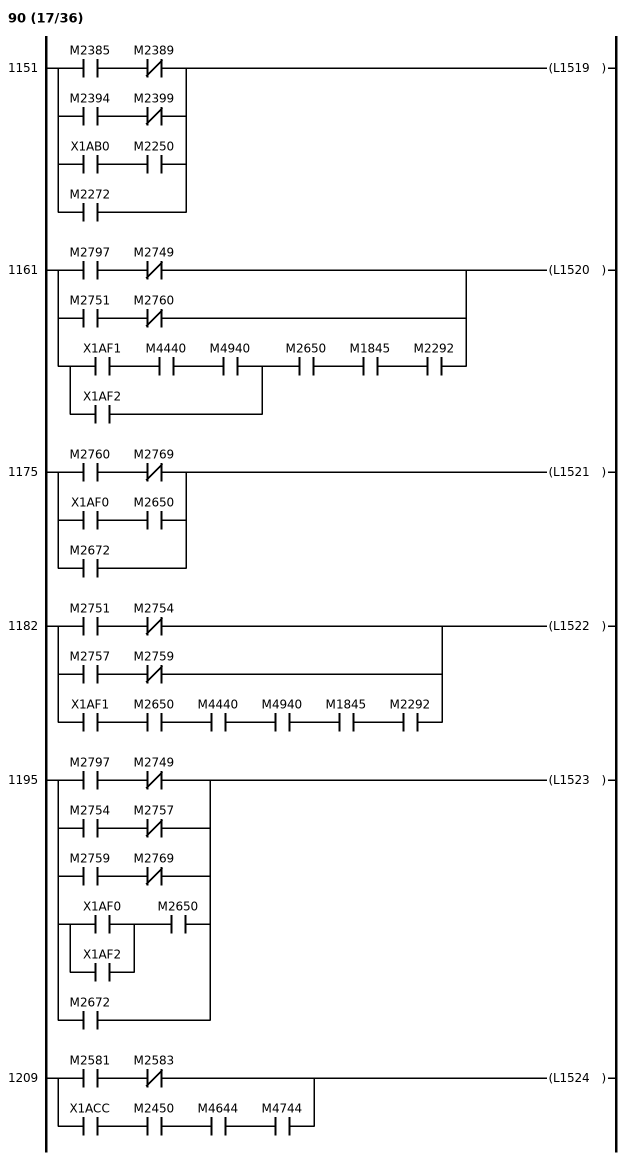
1151  LD      M2385
      ANI     M2389
      LD      M2394
      ANI     M2399
      ORB
      LD      X1AB0
      AND     M2250
      ORB
      OR      M2272
      OUT     L1519
1161  LD      M2797
      ANI     M2749
      LD      M2751
      ANI     M2760
      ORB
      LD      X1AF1
      AND     M4440
      AND     M4940
      OR      X1AF2
      AND     M2650
      AND     M1845
      AND     M2292
      ORB
      OUT     L1520
1175  LD      M2760
      ANI     M2769
      LD      X1AF0
      AND     M2650
      ORB
      OR      M2672
      OUT     L1521
1182  LD      M2751
      ANI     M2754
      LD      M2757
      ANI     M2759
      ORB
      LD      X1AF1
      AND     M2650
      AND     M4440
      AND     M4940
      AND     M1845
      AND     M2292
      ORB
      OUT     L1522
1195  LD      M2797
      ANI     M2749
      LD      M2754
      ANI     M2757
      ORB
      LD      M2759
      ANI     M2769
      ORB
      LD      X1AF0
      OR      X1AF2
      AND     M2650
      ORB
      OR      M2672
      OUT     L1523
1209  LD      M2581
      ANI     M2583
      LD      X1ACC
      AND     M2450
      AND     M4644
      AND     M4744
      ORB
      OUT     L1524
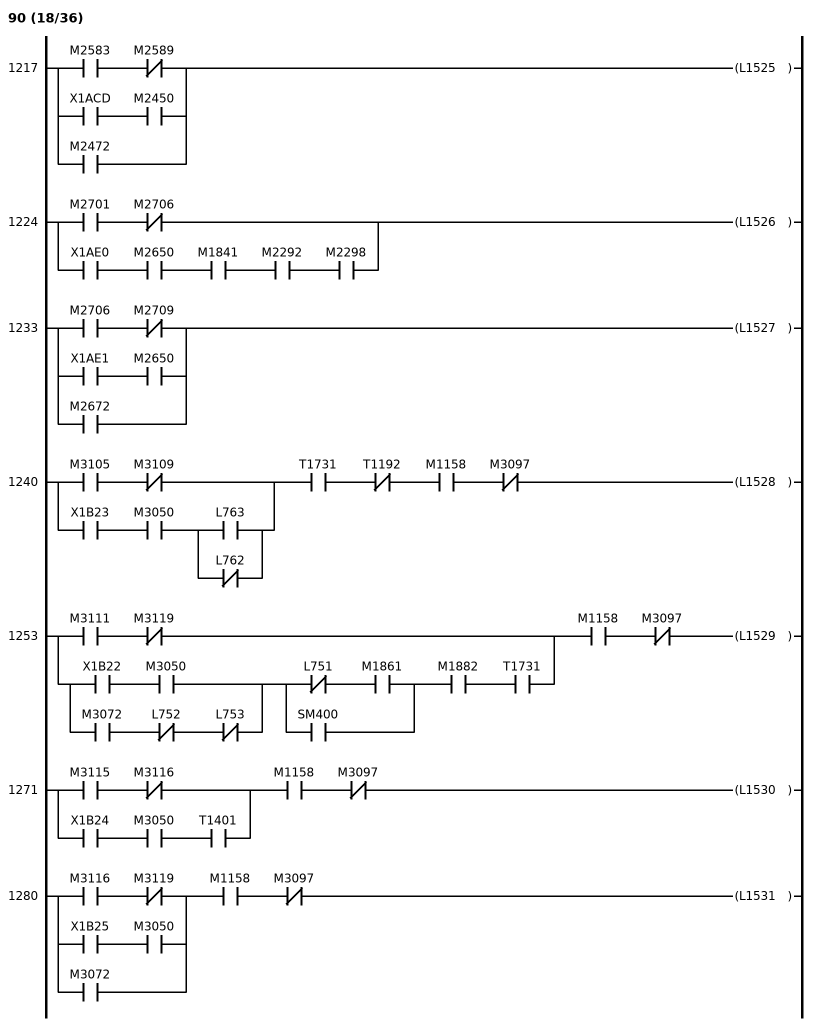
1217  LD      M2583
      ANI     M2589
      LD      X1ACD
      AND     M2450
      ORB
      OR      M2472
      OUT     L1525
1224  LD      M2701
      ANI     M2706
      LD      X1AE0
      AND     M2650
      AND     M1841
      AND     M2292
      AND     M2298
      ORB
      OUT     L1526
1233  LD      M2706
      ANI     M2709
      LD      X1AE1
      AND     M2650
      ORB
      OR      M2672
      OUT     L1527
1240  LD      M3105
      ANI     M3109
      LD      X1B23
      AND     M3050
      LD      L763
      ORI     L762
      ANB
      ORB
      AND     T1731
      ANI     T1192
      AND     M1158
      ANI     M3097
      OUT     L1528
1253  LD      M3111
      ANI     M3119
      LD      X1B22
      AND     M3050
      LD      M3072
      ANI     L752
      ANI     L753
      ORB
      LDI     L751
      AND     M1861
      OR      SM400
      ANB
      AND     M1882
      AND     T1731
      ORB
      AND     M1158
      ANI     M3097
      OUT     L1529
1271  LD      M3115
      ANI     M3116
      LD      X1B24
      AND     M3050
      AND     T1401
      ORB
      AND     M1158
      ANI     M3097
      OUT     L1530
1280  LD      M3116
      ANI     M3119
      LD      X1B25
      AND     M3050
      ORB
      OR      M3072
      AND     M1158
      ANI     M3097
      OUT     L1531
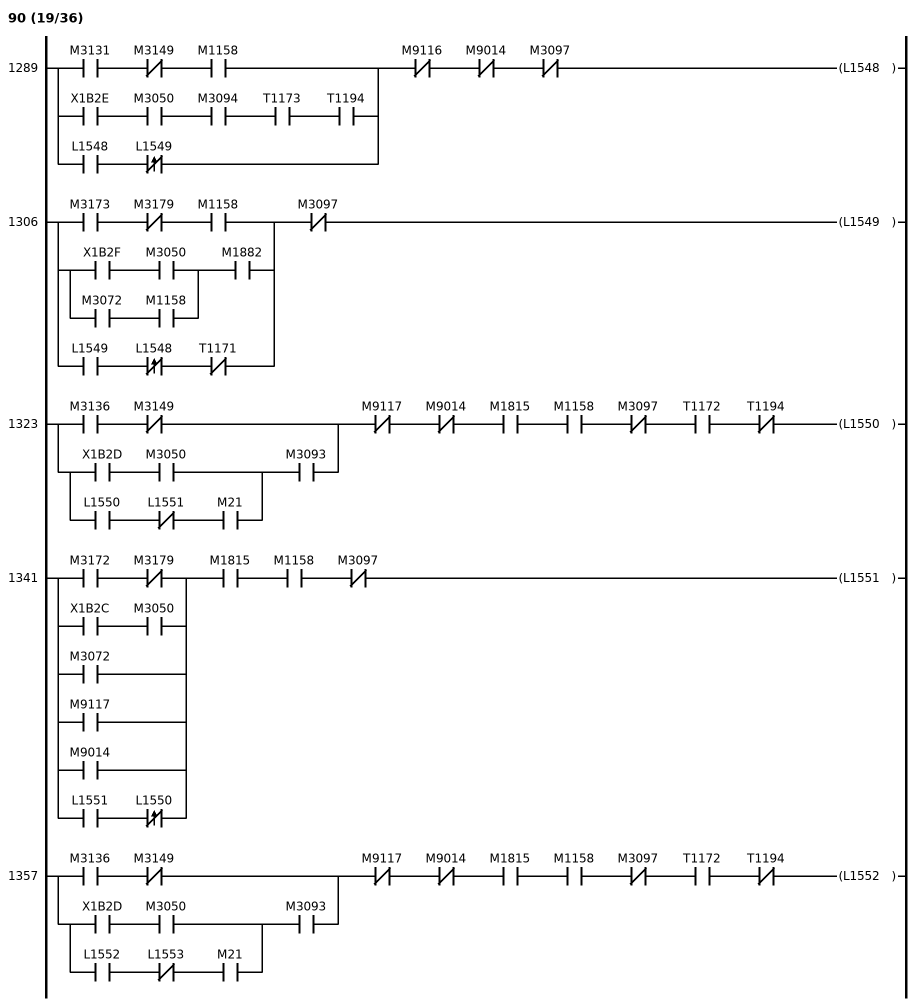
1289  LD      M3131
      ANI     M3149
      AND     M1158
      LD      X1B2E
      AND     M3050
      AND     M3094
      AND     T1173
      AND     T1194
      ORB
      LD      L1548
      ANDPI   L1549
      ORB
      ANI     M9116
      ANI     M9014
      ANI     M3097
      OUT     L1548
1306  LD      M3173
      ANI     M3179
      AND     M1158
      LD      X1B2F
      AND     M3050
      LD      M3072
      AND     M1158
      ORB
      AND     M1882
      ORB
      LD      L1549
      ANDPI   L1548
      ANI     T1171
      ORB
      ANI     M3097
      OUT     L1549
1323  LD      M3136
      ANI     M3149
      LD      X1B2D
      AND     M3050
      LD      L1550
      ANI     L1551
      AND     M21
      ORB
      AND     M3093
      ORB
      ANI     M9117
      ANI     M9014
      AND     M1815
      AND     M1158
      ANI     M3097
      AND     T1172
      ANI     T1194
      OUT     L1550
1341  LD      M3172
      ANI     M3179
      LD      X1B2C
      AND     M3050
      ORB
      OR      M3072
      OR      M9117
      OR      M9014
      LD      L1551
      ANDPI   L1550
      ORB
      AND     M1815
      AND     M1158
      ANI     M3097
      OUT     L1551
1357  LD      M3136
      ANI     M3149
      LD      X1B2D
      AND     M3050
      LD      L1552
      ANI     L1553
      AND     M21
      ORB
      AND     M3093
      ORB
      ANI     M9117
      ANI     M9014
      AND     M1815
      AND     M1158
      ANI     M3097
      AND     T1172
      ANI     T1194
      OUT     L1552
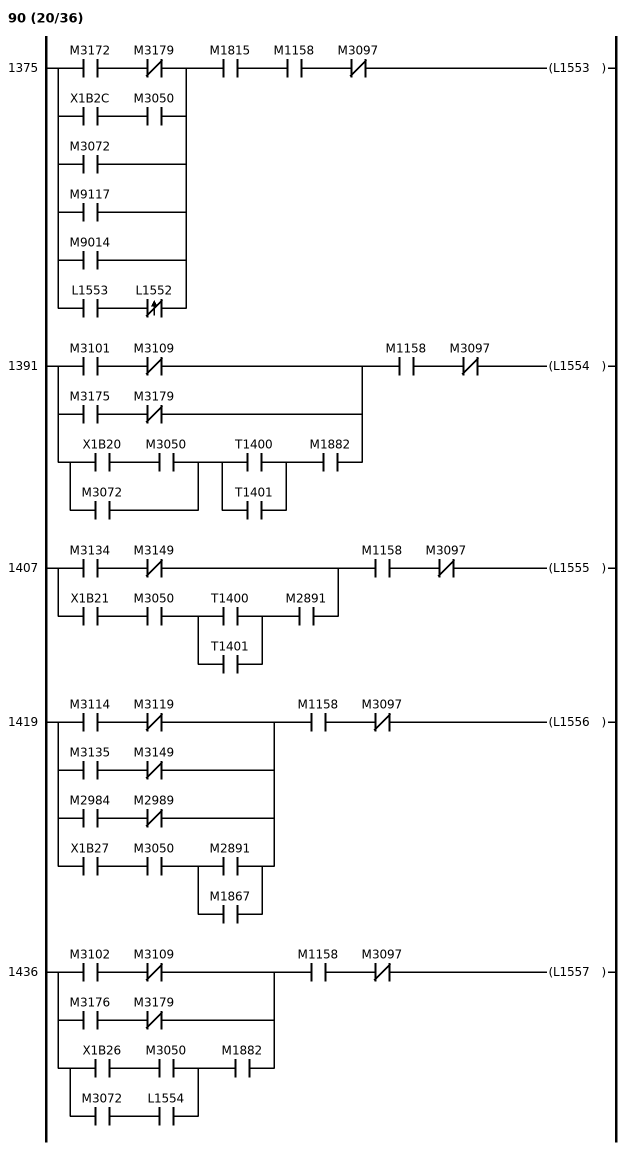
1375  LD      M3172
      ANI     M3179
      LD      X1B2C
      AND     M3050
      ORB
      OR      M3072
      OR      M9117
      OR      M9014
      LD      L1553
      ANDPI   L1552
      ORB
      AND     M1815
      AND     M1158
      ANI     M3097
      OUT     L1553
1391  LD      M3101
      ANI     M3109
      LD      M3175
      ANI     M3179
      ORB
      LD      X1B20
      AND     M3050
      OR      M3072
      LD      T1400
      OR      T1401
      ANB
      AND     M1882
      ORB
      AND     M1158
      ANI     M3097
      OUT     L1554
1407  LD      M3134
      ANI     M3149
      LD      X1B21
      AND     M3050
      LD      T1400
      OR      T1401
      ANB
      AND     M2891
      ORB
      AND     M1158
      ANI     M3097
      OUT     L1555
1419  LD      M3114
      ANI     M3119
      LD      M3135
      ANI     M3149
      ORB
      LD      M2984
      ANI     M2989
      ORB
      LD      X1B27
      AND     M3050
      LD      M2891
      OR      M1867
      ANB
      ORB
      AND     M1158
      ANI     M3097
      OUT     L1556
1436  LD      M3102
      ANI     M3109
      LD      M3176
      ANI     M3179
      ORB
      LD      X1B26
      AND     M3050
      LD      M3072
      AND     L1554
      ORB
      AND     M1882
      ORB
      AND     M1158
      ANI     M3097
      OUT     L1557
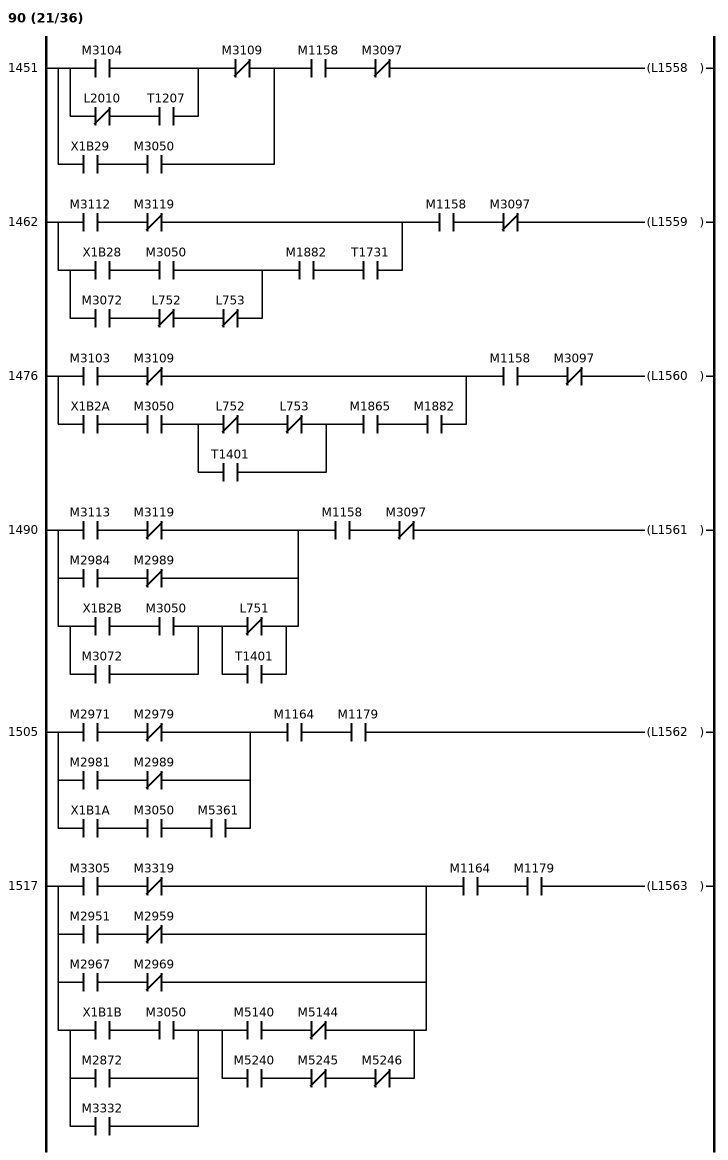
1451  LD      M3104
      LDI     L2010
      AND     T1207
      ORB
      ANI     M3109
      LD      X1B29
      AND     M3050
      ORB
      AND     M1158
      ANI     M3097
      OUT     L1558
1462  LD      M3112
      ANI     M3119
      LD      X1B28
      AND     M3050
      LD      M3072
      ANI     L752
      ANI     L753
      ORB
      AND     M1882
      AND     T1731
      ORB
      AND     M1158
      ANI     M3097
      OUT     L1559
1476  LD      M3103
      ANI     M3109
      LD      X1B2A
      AND     M3050
      LDI     L752
      ANI     L753
      OR      T1401
      ANB
      AND     M1865
      AND     M1882
      ORB
      AND     M1158
      ANI     M3097
      OUT     L1560
1490  LD      M3113
      ANI     M3119
      LD      M2984
      ANI     M2989
      ORB
      LD      X1B2B
      AND     M3050
      OR      M3072
      LDI     L751
      OR      T1401
      ANB
      ORB
      AND     M1158
      ANI     M3097
      OUT     L1561
1505  LD      M2971
      ANI     M2979
      LD      M2981
      ANI     M2989
      ORB
      LD      X1B1A
      AND     M3050
      AND     M5361
      ORB
      AND     M1164
      AND     M1179
      OUT     L1562
1517  LD      M3305
      ANI     M3319
      LD      M2951
      ANI     M2959
      ORB
      LD      M2967
      ANI     M2969
      ORB
      LD      X1B1B
      AND     M3050
      OR      M2872
      OR      M3332
      LD      M5140
      ANI     M5144
      LD      M5240
      ANI     M5245
      ANI     M5246
      ORB
      ANB
      ORB
      AND     M1164
      AND     M1179
      OUT     L1563
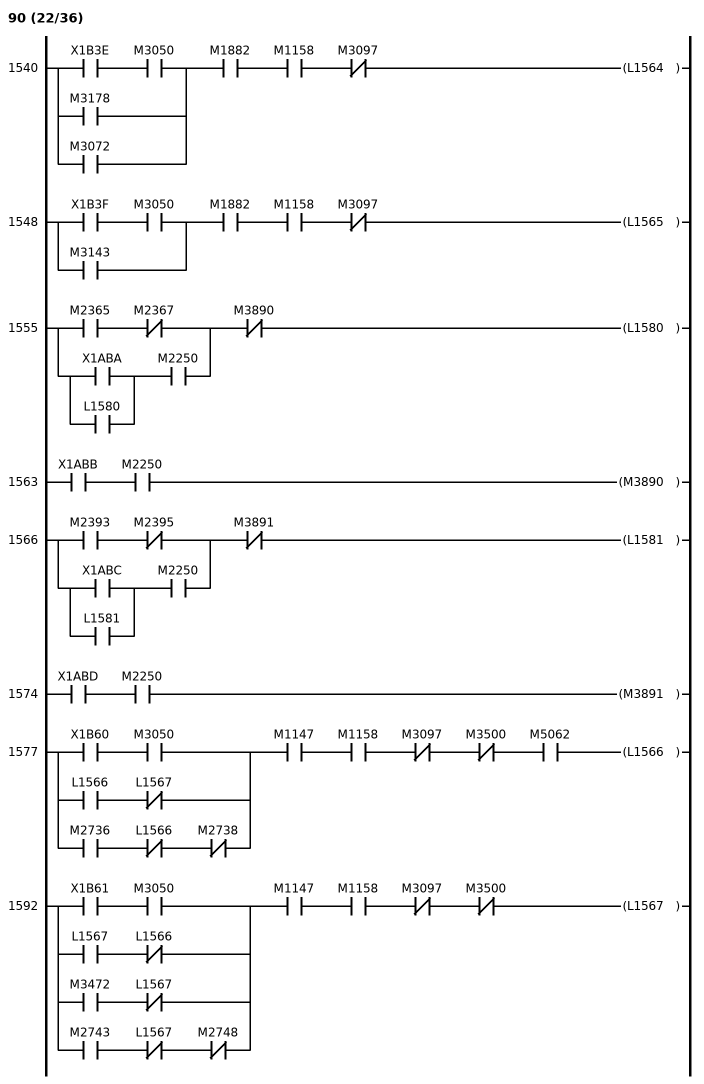
1540  LD      X1B3E
      AND     M3050
      OR      M3178
      OR      M3072
      AND     M1882
      AND     M1158
      ANI     M3097
      OUT     L1564
1548  LD      X1B3F
      AND     M3050
      OR      M3143
      AND     M1882
      AND     M1158
      ANI     M3097
      OUT     L1565
1555  LD      M2365
      ANI     M2367
      LD      X1ABA
      OR      L1580
      AND     M2250
      ORB
      ANI     M3890
      OUT     L1580
1563  LD      X1ABB
      AND     M2250
      OUT     M3890
1566  LD      M2393
      ANI     M2395
      LD      X1ABC
      OR      L1581
      AND     M2250
      ORB
      ANI     M3891
      OUT     L1581
1574  LD      X1ABD
      AND     M2250
      OUT     M3891
1577  LD      X1B60
      AND     M3050
      LD      L1566
      ANI     L1567
      ORB
      LD      M2736
      ANI     L1566
      ANI     M2738
      ORB
      AND     M1147
      AND     M1158
      ANI     M3097
      ANI     M3500
      AND     M5062
      OUT     L1566
1592  LD      X1B61
      AND     M3050
      LD      L1567
      ANI     L1566
      ORB
      LD      M3472
      ANI     L1567
      ORB
      LD      M2743
      ANI     L1567
      ANI     M2748
      ORB
      AND     M1147
      AND     M1158
      ANI     M3097
      ANI     M3500
      OUT     L1567
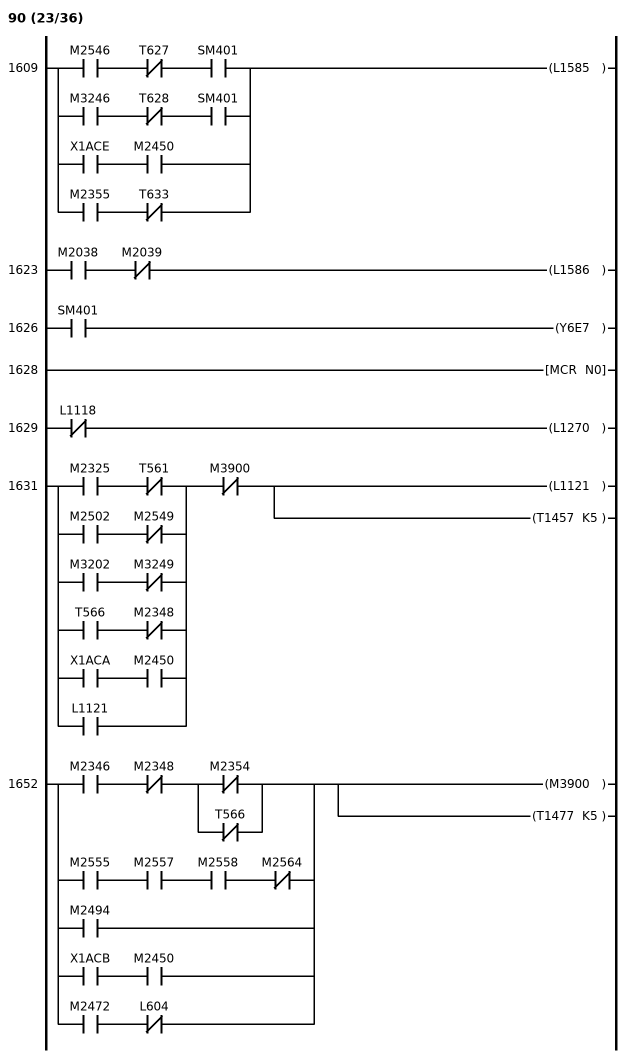
1609  LD      M2546
      ANI     T627
      AND     SM401
      LD      M3246
      ANI     T628
      AND     SM401
      ORB
      LD      X1ACE
      AND     M2450
      ORB
      LD      M2355
      ANI     T633
      ORB
      OUT     L1585
1623  LD      M2038
      ANI     M2039
      OUT     L1586
1626  LD      SM401
      OUT     Y6E7
1628  MCR     N0
1629  LDI     L1118
      OUT     L1270
1631  LD      M2325
      ANI     T561
      LD      M2502
      ANI     M2549
      ORB
      LD      M3202
      ANI     M3249
      ORB
      LD      T566
      ANI     M2348
      ORB
      LD      X1ACA
      AND     M2450
      ORB
      OR      L1121
      ANI     M3900
      OUT     L1121
      OUT     T1457 K5
1652  LD      M2346
      ANI     M2348
      LDI     M2354
      ORI     T566
      ANB
      LD      M2555
      AND     M2557
      AND     M2558
      ANI     M2564
      ORB
      OR      M2494
      LD      X1ACB
      AND     M2450
      ORB
      LD      M2472
      ANI     L604
      ORB
      OUT     M3900
      OUT     T1477 K5
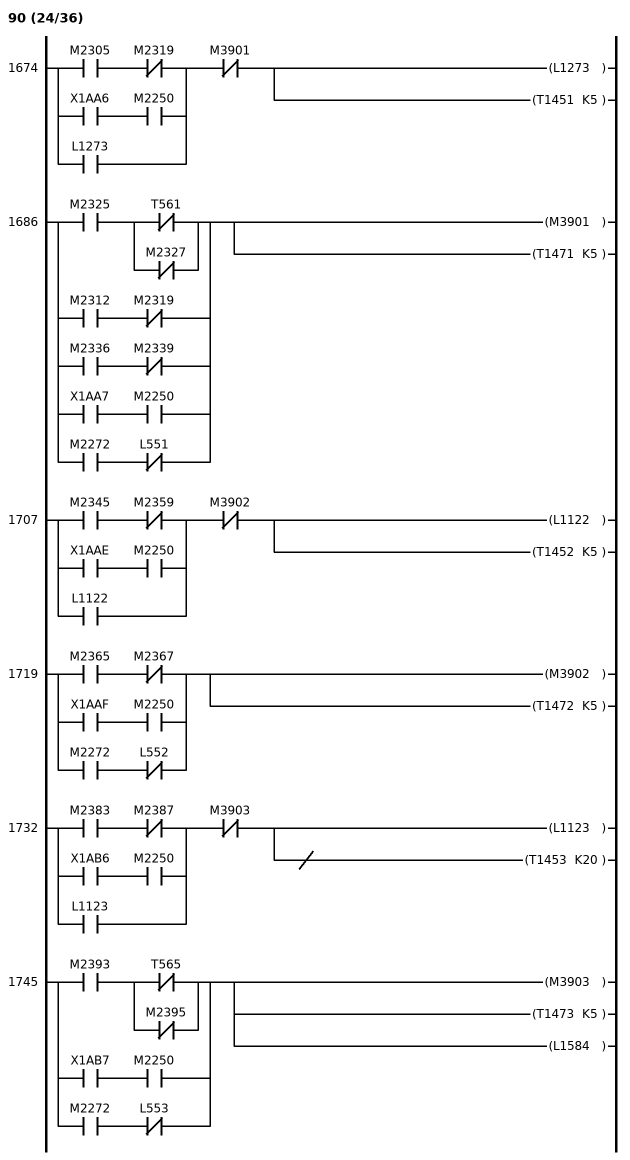
1674  LD      M2305
      ANI     M2319
      LD      X1AA6
      AND     M2250
      ORB
      OR      L1273
      ANI     M3901
      OUT     L1273
      OUT     T1451 K5
1686  LD      M2325
      LDI     T561
      ORI     M2327
      ANB
      LD      M2312
      ANI     M2319
      ORB
      LD      M2336
      ANI     M2339
      ORB
      LD      X1AA7
      AND     M2250
      ORB
      LD      M2272
      ANI     L551
      ORB
      OUT     M3901
      OUT     T1471 K5
1707  LD      M2345
      ANI     M2359
      LD      X1AAE
      AND     M2250
      ORB
      OR      L1122
      ANI     M3902
      OUT     L1122
      OUT     T1452 K5
1719  LD      M2365
      ANI     M2367
      LD      X1AAF
      AND     M2250
      ORB
      LD      M2272
      ANI     L552
      ORB
      OUT     M3902
      OUT     T1472 K5
1732  LD      M2383
      ANI     M2387
      LD      X1AB6
      AND     M2250
      ORB
      OR      L1123
      ANI     M3903
      OUT     L1123
      INV
      OUT     T1453 K20
1745  LD      M2393
      LDI     T565
      ORI     M2395
      ANB
      LD      X1AB7
      AND     M2250
      ORB
      LD      M2272
      ANI     L553
      ORB
      OUT     M3903
      OUT     T1473 K5
      OUT     L1584
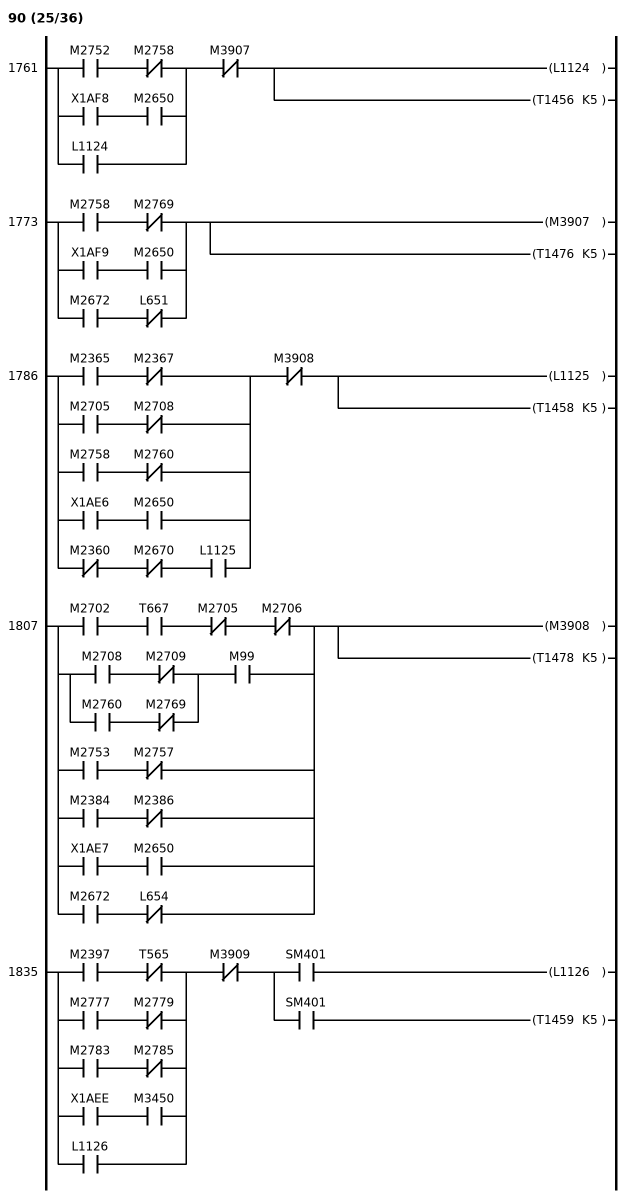
1761  LD      M2752
      ANI     M2758
      LD      X1AF8
      AND     M2650
      ORB
      OR      L1124
      ANI     M3907
      OUT     L1124
      OUT     T1456 K5
1773  LD      M2758
      ANI     M2769
      LD      X1AF9
      AND     M2650
      ORB
      LD      M2672
      ANI     L651
      ORB
      OUT     M3907
      OUT     T1476 K5
1786  LD      M2365
      ANI     M2367
      LD      M2705
      ANI     M2708
      ORB
      LD      M2758
      ANI     M2760
      ORB
      LD      X1AE6
      AND     M2650
      ORB
      LDI     M2360
      ANI     M2670
      AND     L1125
      ORB
      ANI     M3908
      OUT     L1125
      OUT     T1458 K5
1807  LD      M2702
      AND     T667
      ANI     M2705
      ANI     M2706
      LD      M2708
      ANI     M2709
      LD      M2760
      ANI     M2769
      ORB
      AND     M99
      ORB
      LD      M2753
      ANI     M2757
      ORB
      LD      M2384
      ANI     M2386
      ORB
      LD      X1AE7
      AND     M2650
      ORB
      LD      M2672
      ANI     L654
      ORB
      OUT     M3908
      OUT     T1478 K5
1835  LD      M2397
      ANI     T565
      LD      M2777
      ANI     M2779
      ORB
      LD      M2783
      ANI     M2785
      ORB
      LD      X1AEE
      AND     M3450
      ORB
      OR      L1126
      ANI     M3909
      MPS
      AND     SM401
      OUT     L1126
      MPP
      AND     SM401
      OUT     T1459 K5
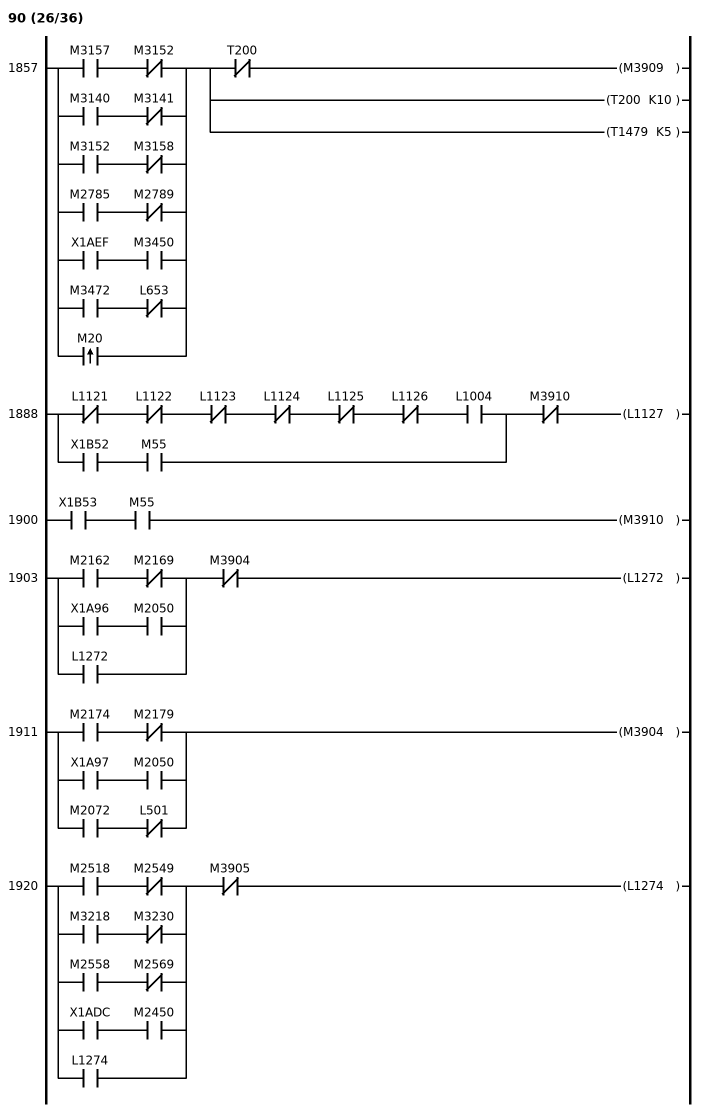
1857  LD      M3157
      ANI     M3152
      LD      M3140
      ANI     M3141
      ORB
      LD      M3152
      ANI     M3158
      ORB
      LD      M2785
      ANI     M2789
      ORB
      LD      X1AEF
      AND     M3450
      ORB
      LD      M3472
      ANI     L653
      ORB
      ORP     M20
      MPS
      ANI     T200
      OUT     M3909
      MPP
      OUT     T200 K10
      OUT     T1479 K5
1888  LDI     L1121
      ANI     L1122
      ANI     L1123
      ANI     L1124
      ANI     L1125
      ANI     L1126
      AND     L1004
      LD      X1B52
      AND     M55
      ORB
      ANI     M3910
      OUT     L1127
1900  LD      X1B53
      AND     M55
      OUT     M3910
1903  LD      M2162
      ANI     M2169
      LD      X1A96
      AND     M2050
      ORB
      OR      L1272
      ANI     M3904
      OUT     L1272
1911  LD      M2174
      ANI     M2179
      LD      X1A97
      AND     M2050
      ORB
      LD      M2072
      ANI     L501
      ORB
      OUT     M3904
1920  LD      M2518
      ANI     M2549
      LD      M3218
      ANI     M3230
      ORB
      LD      M2558
      ANI     M2569
      ORB
      LD      X1ADC
      AND     M2450
      ORB
      OR      L1274
      ANI     M3905
      OUT     L1274
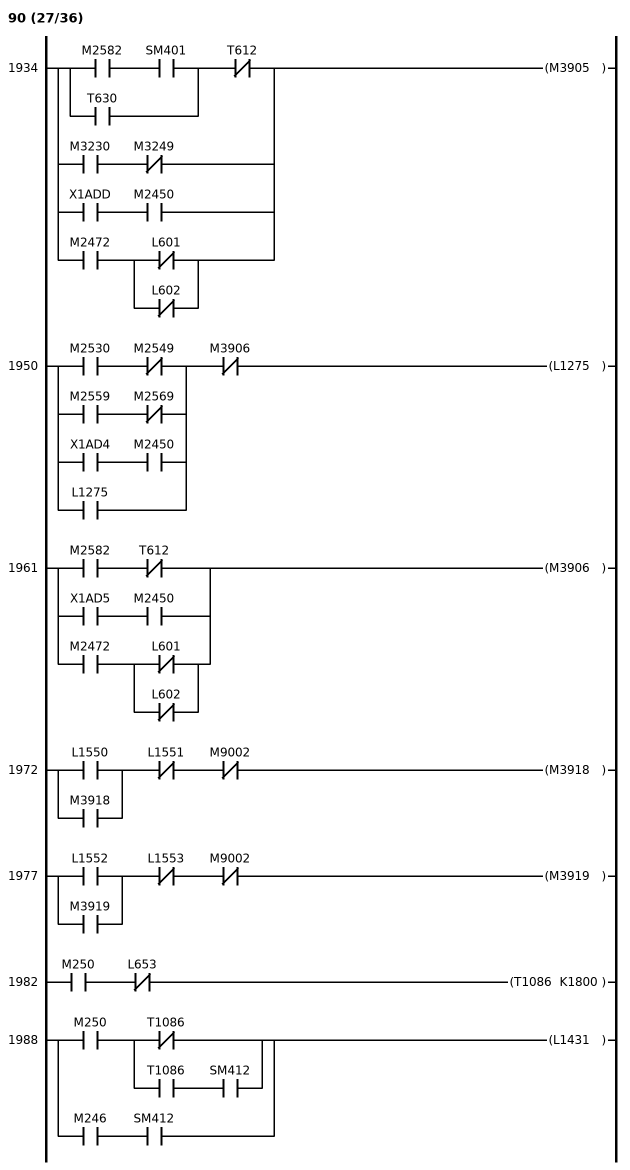
1934  LD      M2582
      AND     SM401
      OR      T630
      ANI     T612
      LD      M3230
      ANI     M3249
      ORB
      LD      X1ADD
      AND     M2450
      ORB
      LD      M2472
      LDI     L601
      ORI     L602
      ANB
      ORB
      OUT     M3905
1950  LD      M2530
      ANI     M2549
      LD      M2559
      ANI     M2569
      ORB
      LD      X1AD4
      AND     M2450
      ORB
      OR      L1275
      ANI     M3906
      OUT     L1275
1961  LD      M2582
      ANI     T612
      LD      X1AD5
      AND     M2450
      ORB
      LD      M2472
      LDI     L601
      ORI     L602
      ANB
      ORB
      OUT     M3906
1972  LD      L1550
      OR      M3918
      ANI     L1551
      ANI     M9002
      OUT     M3918
1977  LD      L1552
      OR      M3919
      ANI     L1553
      ANI     M9002
      OUT     M3919
1982  LD      M250
      ANI     L653
      OUT     T1086 K1800
1988  LD      M250
      LDI     T1086
      LD      T1086
      AND     SM412
      ORB
      ANB
      LD      M246
      AND     SM412
      ORB
      OUT     L1431
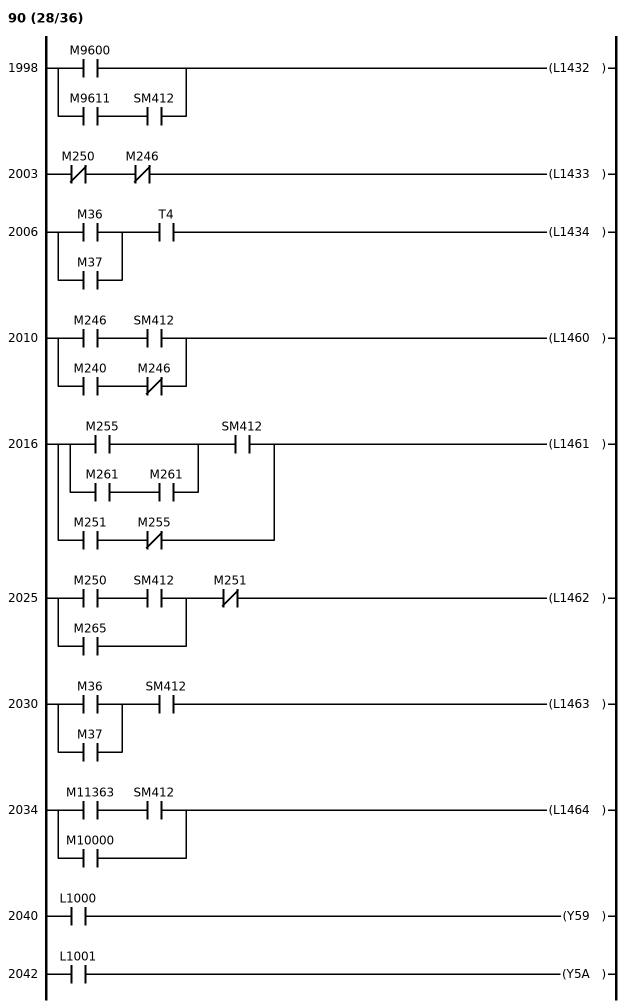
1998  LD      M9600
      LD      M9611
      AND     SM412
      ORB
      OUT     L1432
2003  LDI     M250
      ANI     M246
      OUT     L1433
2006  LD      M36
      OR      M37
      AND     T4
      OUT     L1434
2010  LD      M246
      AND     SM412
      LD      M240
      ANI     M246
      ORB
      OUT     L1460
2016  LD      M255
      LD      M261
      AND     M261
      ORB
      AND     SM412
      LD      M251
      ANI     M255
      ORB
      OUT     L1461
2025  LD      M250
      AND     SM412
      OR      M265
      ANI     M251
      OUT     L1462
2030  LD      M36
      OR      M37
      AND     SM412
      OUT     L1463
2034  LD      M11363
      AND     SM412
      OR      M10000
      OUT     L1464
; 
2040  LD      L1000
      OUT     Y59
2042  LD      L1001
      OUT     Y5A
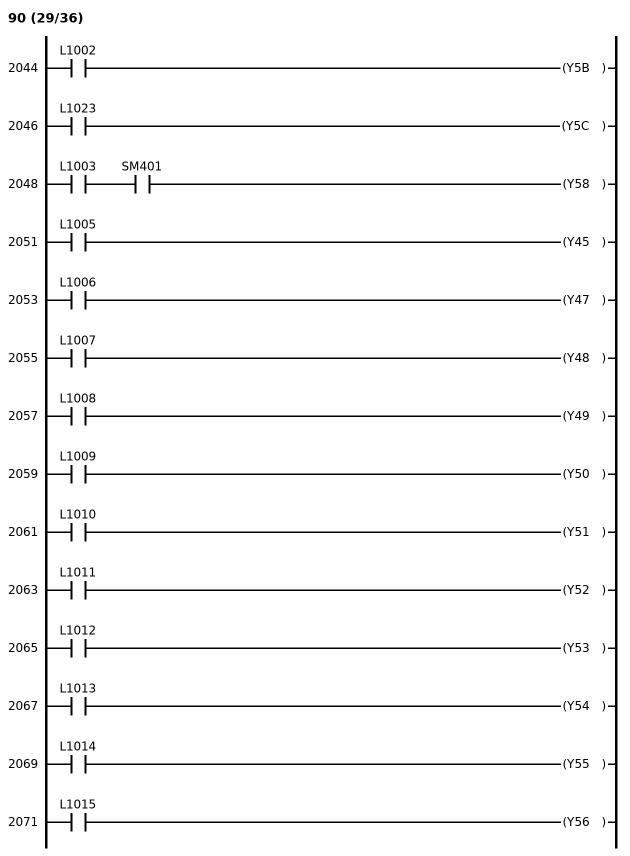
2044  LD      L1002
      OUT     Y5B
2046  LD      L1023
      OUT     Y5C
2048  LD      L1003
      AND     SM401
      OUT     Y58
2051  LD      L1005
      OUT     Y45
2053  LD      L1006
      OUT     Y47
2055  LD      L1007
      OUT     Y48
2057  LD      L1008
      OUT     Y49
2059  LD      L1009
      OUT     Y50
2061  LD      L1010
      OUT     Y51
2063  LD      L1011
      OUT     Y52
2065  LD      L1012
      OUT     Y53
2067  LD      L1013
      OUT     Y54
2069  LD      L1014
      OUT     Y55
2071  LD      L1015
      OUT     Y56
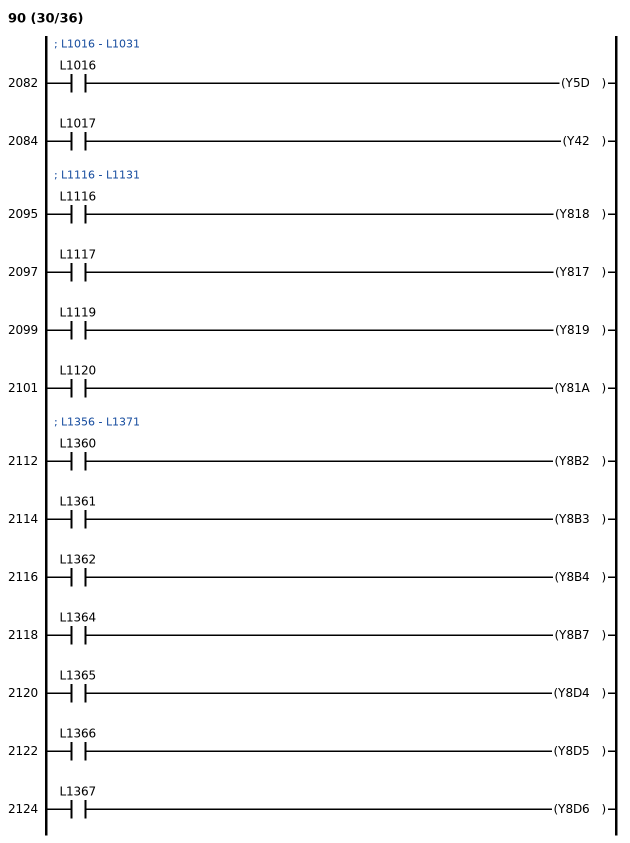
; L1016 - L1031
2082  LD      L1016
      OUT     Y5D
2084  LD      L1017
      OUT     Y42
; L1116 - L1131
2095  LD      L1116
      OUT     Y818
2097  LD      L1117
      OUT     Y817
2099  LD      L1119
      OUT     Y819
2101  LD      L1120
      OUT     Y81A
; L1356 - L1371
2112  LD      L1360
      OUT     Y8B2
2114  LD      L1361
      OUT     Y8B3
2116  LD      L1362
      OUT     Y8B4
2118  LD      L1364
      OUT     Y8B7
2120  LD      L1365
      OUT     Y8D4
2122  LD      L1366
      OUT     Y8D5
2124  LD      L1367
      OUT     Y8D6
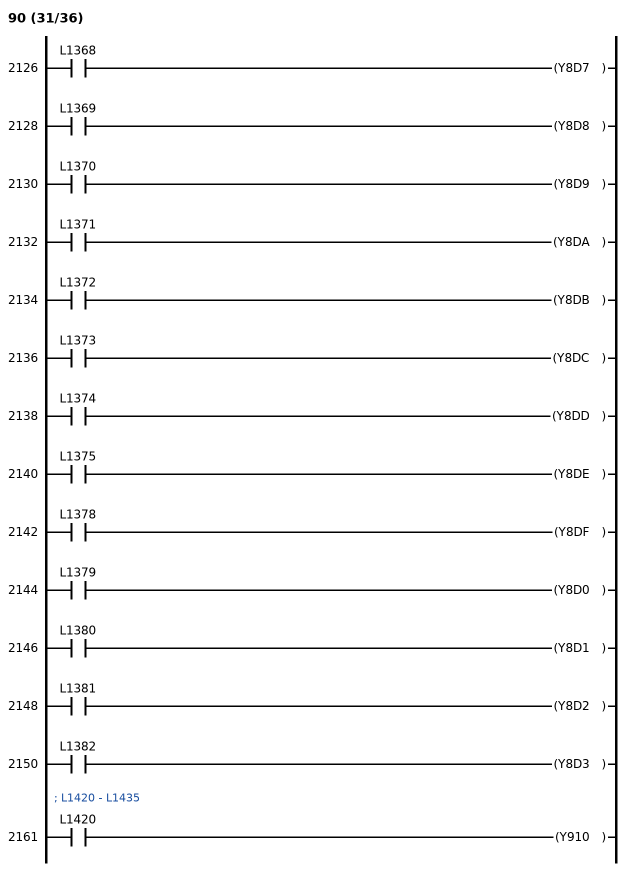
2126  LD      L1368
      OUT     Y8D7
2128  LD      L1369
      OUT     Y8D8
2130  LD      L1370
      OUT     Y8D9
2132  LD      L1371
      OUT     Y8DA
2134  LD      L1372
      OUT     Y8DB
2136  LD      L1373
      OUT     Y8DC
2138  LD      L1374
      OUT     Y8DD
2140  LD      L1375
      OUT     Y8DE
2142  LD      L1378
      OUT     Y8DF
2144  LD      L1379
      OUT     Y8D0
2146  LD      L1380
      OUT     Y8D1
2148  LD      L1381
      OUT     Y8D2
2150  LD      L1382
      OUT     Y8D3
; L1420 - L1435
2161  LD      L1420
      OUT     Y910
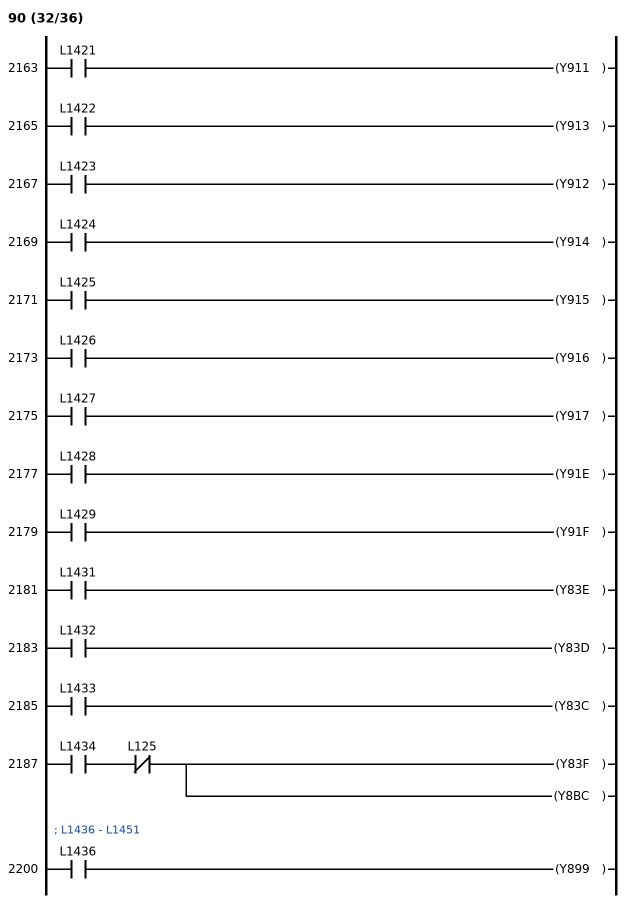
2163  LD      L1421
      OUT     Y911
2165  LD      L1422
      OUT     Y913
2167  LD      L1423
      OUT     Y912
2169  LD      L1424
      OUT     Y914
2171  LD      L1425
      OUT     Y915
2173  LD      L1426
      OUT     Y916
2175  LD      L1427
      OUT     Y917
2177  LD      L1428
      OUT     Y91E
2179  LD      L1429
      OUT     Y91F
2181  LD      L1431
      OUT     Y83E
2183  LD      L1432
      OUT     Y83D
2185  LD      L1433
      OUT     Y83C
2187  LD      L1434
      ANI     L125
      OUT     Y83F
      OUT     Y8BC
; L1436 - L1451
2200  LD      L1436
      OUT     Y899
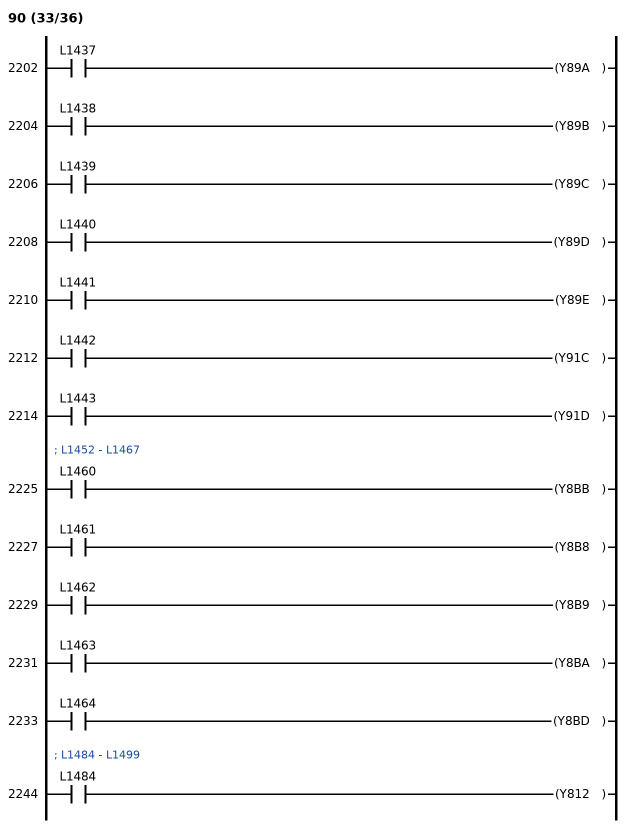
2202  LD      L1437
      OUT     Y89A
2204  LD      L1438
      OUT     Y89B
2206  LD      L1439
      OUT     Y89C
2208  LD      L1440
      OUT     Y89D
2210  LD      L1441
      OUT     Y89E
2212  LD      L1442
      OUT     Y91C
2214  LD      L1443
      OUT     Y91D
; L1452 - L1467
2225  LD      L1460
      OUT     Y8BB
2227  LD      L1461
      OUT     Y8B8
2229  LD      L1462
      OUT     Y8B9
2231  LD      L1463
      OUT     Y8BA
2233  LD      L1464
      OUT     Y8BD
; L1484 - L1499
2244  LD      L1484
      OUT     Y812
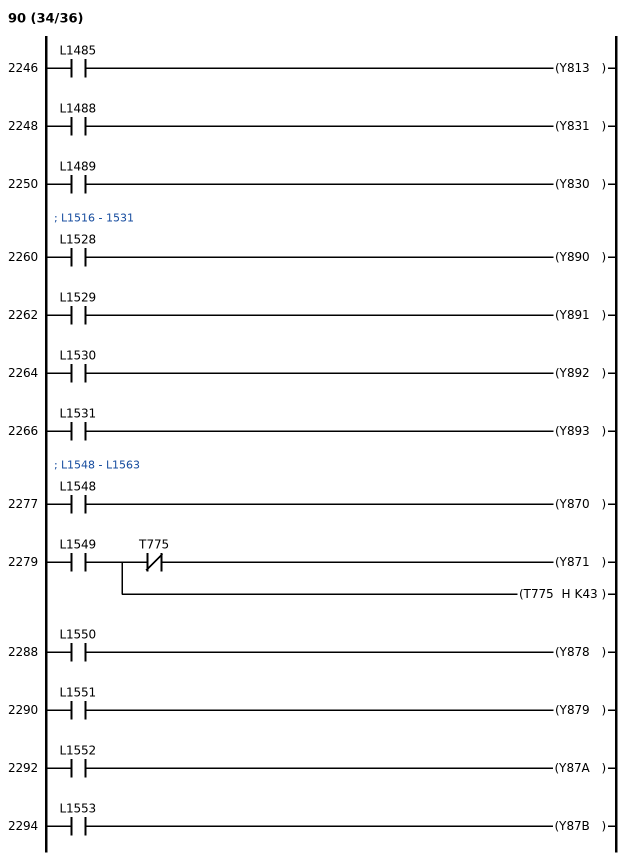
2246  LD      L1485
      OUT     Y813
2248  LD      L1488
      OUT     Y831
2250  LD      L1489
      OUT     Y830
; L1516 - 1531
2260  LD      L1528
      OUT     Y890
2262  LD      L1529
      OUT     Y891
2264  LD      L1530
      OUT     Y892
2266  LD      L1531
      OUT     Y893
; L1548 - L1563
2277  LD      L1548
      OUT     Y870
2279  LD      L1549
      MPS
      ANI     T775
      OUT     Y871
      MPP
      OUTH    T775 K43
2288  LD      L1550
      OUT     Y878
2290  LD      L1551
      OUT     Y879
2292  LD      L1552
      OUT     Y87A
2294  LD      L1553
      OUT     Y87B
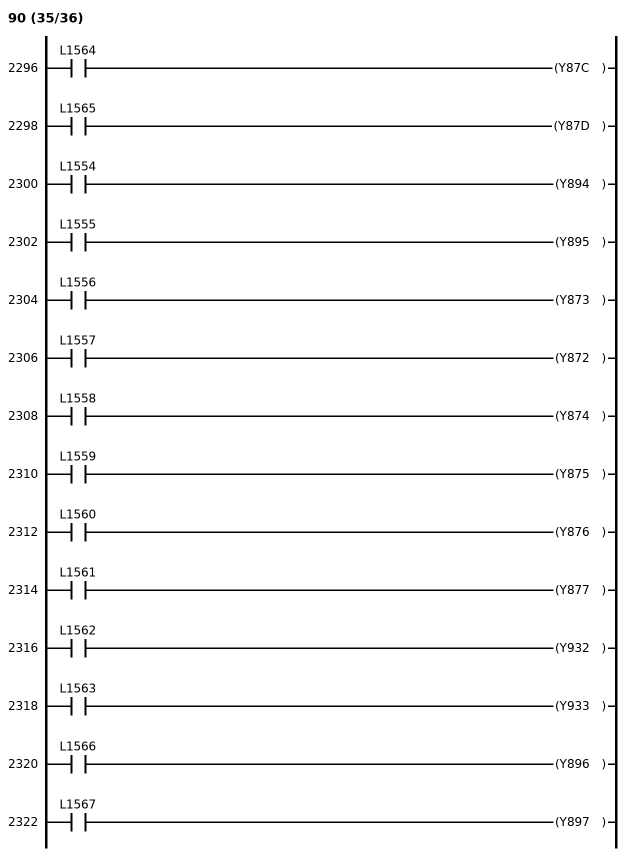
2296  LD      L1564
      OUT     Y87C
2298  LD      L1565
      OUT     Y87D
2300  LD      L1554
      OUT     Y894
2302  LD      L1555
      OUT     Y895
2304  LD      L1556
      OUT     Y873
2306  LD      L1557
      OUT     Y872
2308  LD      L1558
      OUT     Y874
2310  LD      L1559
      OUT     Y875
2312  LD      L1560
      OUT     Y876
2314  LD      L1561
      OUT     Y877
2316  LD      L1562
      OUT     Y932
2318  LD      L1563
      OUT     Y933
2320  LD      L1566
      OUT     Y896
2322  LD      L1567
      OUT     Y897
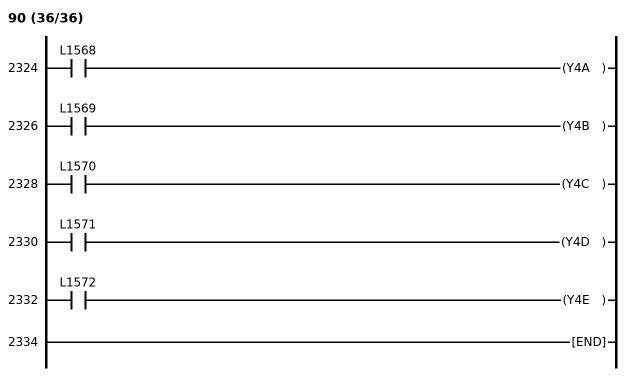
2324  LD      L1568
      OUT     Y4A
2326  LD      L1569
      OUT     Y4B
2328  LD      L1570
      OUT     Y4C
2330  LD      L1571
      OUT     Y4D
2332  LD      L1572
      OUT     Y4E
2334  END
END_PROGRAM

PROGRAM 99
0     END
END_PROGRAM

PROGRAM ADVANCE
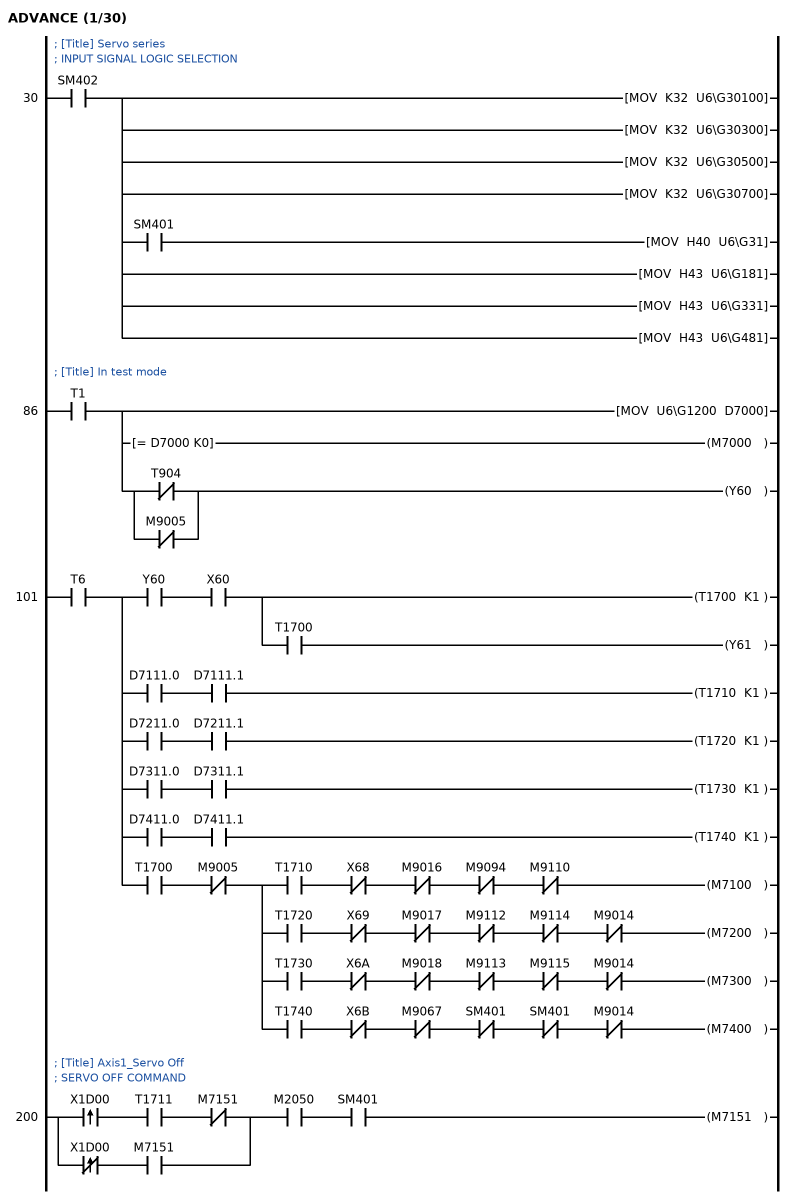
; 
; [Title] Servo series
; INPUT SIGNAL LOGIC SELECTION
; 
30    LD      SM402
      MOV     K32 U6\G30100
      MOV     K32 U6\G30300
      MOV     K32 U6\G30500
      MOV     K32 U6\G30700
      MPS
      AND     SM401
      MOV     H40 U6\G31
      MPP
      MOV     H43 U6\G181
      MOV     H43 U6\G331
      MOV     H43 U6\G481
; 
; 
; 
; [Title] In test mode
; 
; 
; 
; 
86    LD      T1
      MOV     U6\G1200 D7000
      MPS
      AND=    D7000 K0
      OUT     M7000
      MPP
      LDI     T904
      ORI     M9005
      ANB
      OUT     Y60
101   LD      T6
      MPS
      AND     Y60
      AND     X60
      OUT     T1700 K1
      AND     T1700
      OUT     Y61
      MRD
      AND     D7111.0
      AND     D7111.1
      OUT     T1710 K1
      MRD
      AND     D7211.0
      AND     D7211.1
      OUT     T1720 K1
      MRD
      AND     D7311.0
      AND     D7311.1
      OUT     T1730 K1
      MRD
      AND     D7411.0
      AND     D7411.1
      OUT     T1740 K1
      MPP
      AND     T1700
      ANI     M9005
      MPS
      AND     T1710
      ANI     X68
      ANI     M9016
      ANI     M9094
      ANI     M9110
      OUT     M7100
      MRD
      AND     T1720
      ANI     X69
      ANI     M9017
      ANI     M9112
      ANI     M9114
      ANI     M9014
      OUT     M7200
      MRD
      AND     T1730
      ANI     X6A
      ANI     M9018
      ANI     M9113
      ANI     M9115
      ANI     M9014
      OUT     M7300
      MPP
      AND     T1740
      ANI     X6B
      ANI     M9067
      ANI     SM401
      ANI     SM401
      ANI     M9014
      OUT     M7400
; 
; [Title] Axis1_Servo Off
; SERVO OFF COMMAND
; 
200   LDP     X1D00
      AND     T1711
      ANI     M7151
      LDPI    X1D00
      AND     M7151
      ORB
      AND     M2050
      AND     SM401
      OUT     M7151
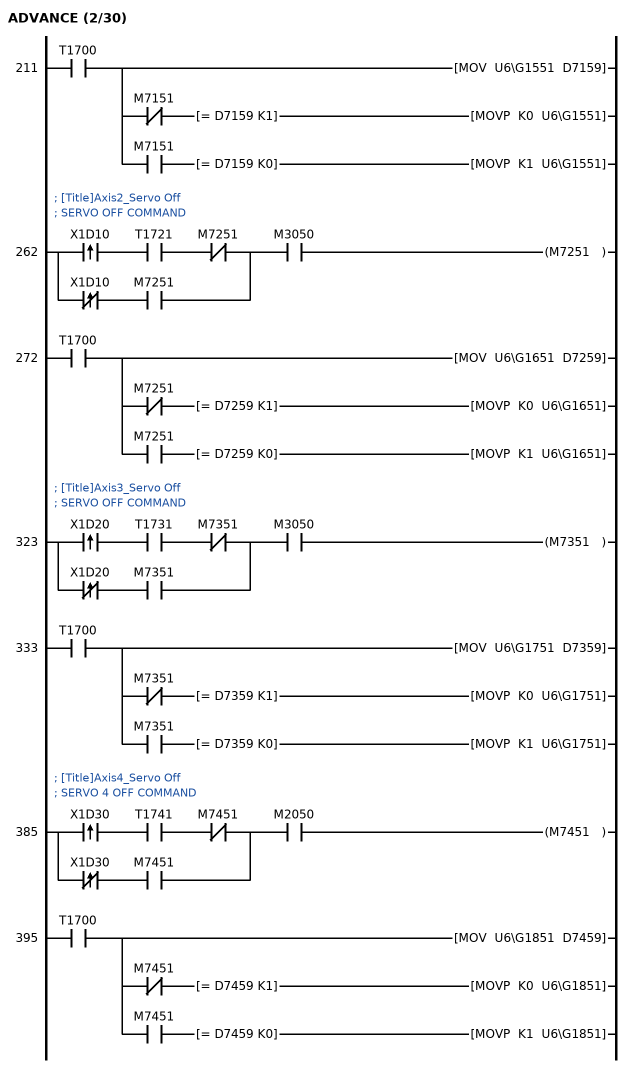
211   LD      T1700
      MOV     U6\G1551 D7159
      MPS
      ANI     M7151
      AND=    D7159 K1
      MOVP    K0 U6\G1551
      MPP
      AND     M7151
      AND=    D7159 K0
      MOVP    K1 U6\G1551
; 
; [Title]Axis2_Servo Off
; SERVO OFF COMMAND
; 
262   LDP     X1D10
      AND     T1721
      ANI     M7251
      LDPI    X1D10
      AND     M7251
      ORB
      AND     M3050
      OUT     M7251
272   LD      T1700
      MOV     U6\G1651 D7259
      MPS
      ANI     M7251
      AND=    D7259 K1
      MOVP    K0 U6\G1651
      MPP
      AND     M7251
      AND=    D7259 K0
      MOVP    K1 U6\G1651
; 
; [Title]Axis3_Servo Off
; SERVO OFF COMMAND
; 
323   LDP     X1D20
      AND     T1731
      ANI     M7351
      LDPI    X1D20
      AND     M7351
      ORB
      AND     M3050
      OUT     M7351
333   LD      T1700
      MOV     U6\G1751 D7359
      MPS
      ANI     M7351
      AND=    D7359 K1
      MOVP    K0 U6\G1751
      MPP
      AND     M7351
      AND=    D7359 K0
      MOVP    K1 U6\G1751
; 
; [Title]Axis4_Servo Off
; SERVO 4 OFF COMMAND
; 
385   LDP     X1D30
      AND     T1741
      ANI     M7451
      LDPI    X1D30
      AND     M7451
      ORB
      AND     M2050
      OUT     M7451
395   LD      T1700
      MOV     U6\G1851 D7459
      MPS
      ANI     M7451
      AND=    D7459 K1
      MOVP    K0 U6\G1851
      MPP
      AND     M7451
      AND=    D7459 K0
      MOVP    K1 U6\G1851
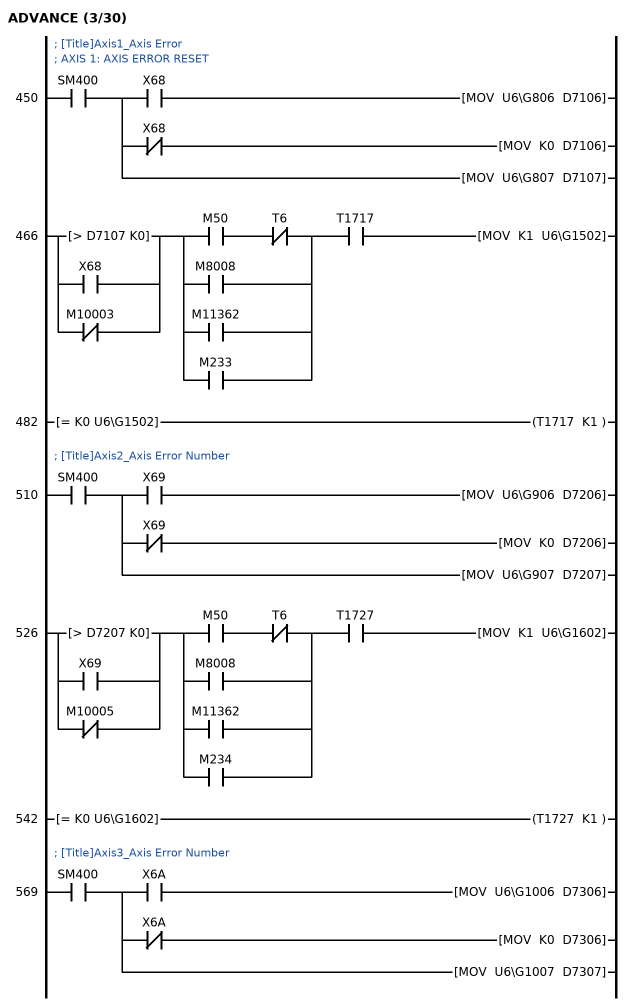
; 
; [Title]Axis1_Axis Error
; AXIS 1: AXIS ERROR RESET
; 
450   LD      SM400
      MPS
      AND     X68
      MOV     U6\G806 D7106
      MRD
      ANI     X68
      MOV     K0 D7106
      MPP
      MOV     U6\G807 D7107
466   LD>     D7107 K0
      OR      X68
      ORI     M10003
      LD      M50
      ANI     T6
      OR      M8008
      OR      M11362
      OR      M233
      ANB
      AND     T1717
      MOV     K1 U6\G1502
482   LD=     K0 U6\G1502
      OUT     T1717 K1
; 
; [Title]Axis2_Axis Error Number
; 
; 
510   LD      SM400
      MPS
      AND     X69
      MOV     U6\G906 D7206
      MRD
      ANI     X69
      MOV     K0 D7206
      MPP
      MOV     U6\G907 D7207
526   LD>     D7207 K0
      OR      X69
      ORI     M10005
      LD      M50
      ANI     T6
      OR      M8008
      OR      M11362
      OR      M234
      ANB
      AND     T1727
      MOV     K1 U6\G1602
542   LD=     K0 U6\G1602
      OUT     T1727 K1
; 
; [Title]Axis3_Axis Error Number
; 
569   LD      SM400
      MPS
      AND     X6A
      MOV     U6\G1006 D7306
      MRD
      ANI     X6A
      MOV     K0 D7306
      MPP
      MOV     U6\G1007 D7307
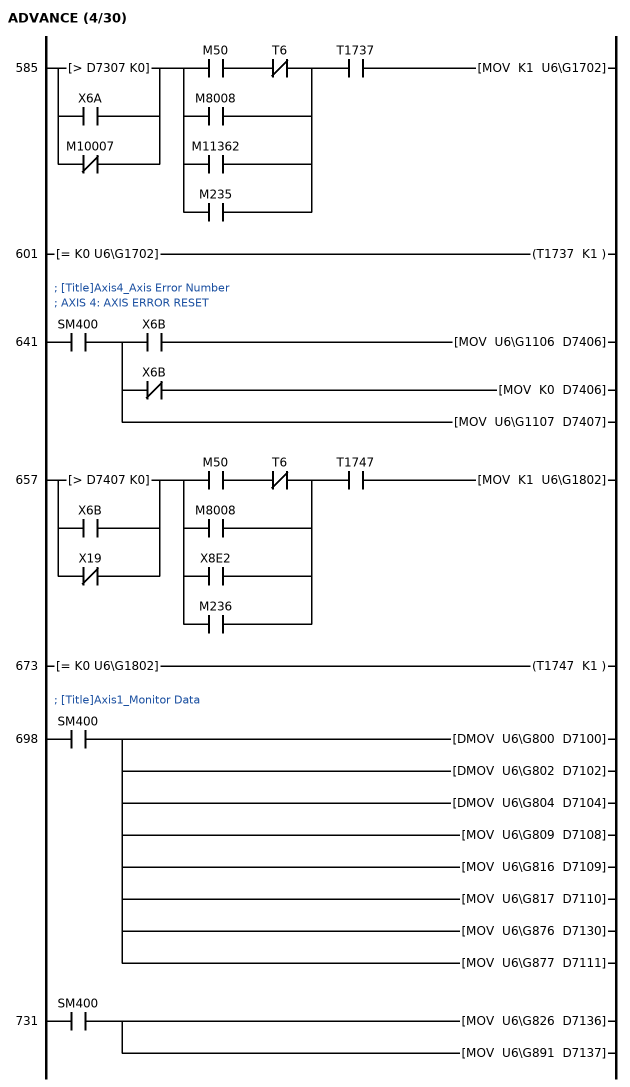
585   LD>     D7307 K0
      OR      X6A
      ORI     M10007
      LD      M50
      ANI     T6
      OR      M8008
      OR      M11362
      OR      M235
      ANB
      AND     T1737
      MOV     K1 U6\G1702
601   LD=     K0 U6\G1702
      OUT     T1737 K1
; 
; [Title]Axis4_Axis Error Number
; AXIS 4: AXIS ERROR RESET
641   LD      SM400
      MPS
      AND     X6B
      MOV     U6\G1106 D7406
      MRD
      ANI     X6B
      MOV     K0 D7406
      MPP
      MOV     U6\G1107 D7407
657   LD>     D7407 K0
      OR      X6B
      ORI     X19
      LD      M50
      ANI     T6
      OR      M8008
      OR      X8E2
      OR      M236
      ANB
      AND     T1747
      MOV     K1 U6\G1802
673   LD=     K0 U6\G1802
      OUT     T1747 K1
; 
; [Title]Axis1_Monitor Data
; 
698   LD      SM400
      DMOV    U6\G800 D7100
      DMOV    U6\G802 D7102
      DMOV    U6\G804 D7104
      MOV     U6\G809 D7108
      MOV     U6\G816 D7109
      MOV     U6\G817 D7110
      MOV     U6\G876 D7130
      MOV     U6\G877 D7111
731   LD      SM400
      MOV     U6\G826 D7136
      MOV     U6\G891 D7137
